% RSLogix 500 project P2a_DIGITAL FILLING STATION STEP METHOD.RSS, saved by version 8.30.00.16 %
PROJECT "PROJECT2"    % processor: Bul.1763 MicroLogix 1100 Series B %

PROGRAM FILES
  LAD 2 "MAIN"  4 rungs
  LAD 3 "IO"  8 rungs  % IO %
  LAD 4 "STEPS"  5 rungs
  LAD 5 "CTRL"  4 rungs

DATA FILES
  O0 OUTPUT  4 elements
  I1 INPUT  6 elements
  S2 STATUS  66 elements
  B3 BINARY  1 elements
  T4 TIMER  1 elements
  C5 COUNTER  1 elements
  R6 CONTROL  1 elements
  N7 INTEGER  1 elements
  F8 FLOAT  1 elements

LADDER 2 "MAIN"
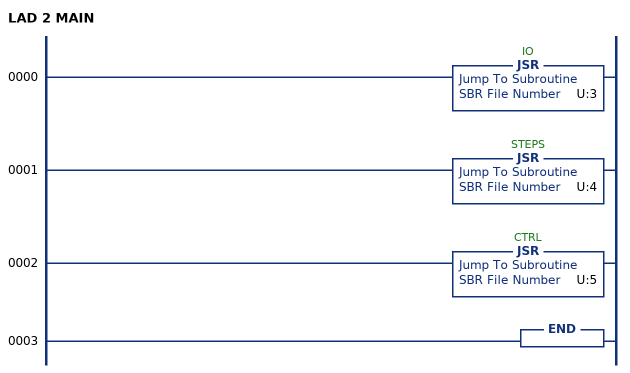
% Rung: 0 %
SOR JSR U:3 EOR
%   U:3  "IO" %
% Rung: 1 %
SOR JSR U:4 EOR
%   U:4  "STEPS" %
% Rung: 2 %
SOR JSR U:5 EOR
%   U:5  "CTRL" %
% Rung: 3 %
SOR END EOR

LADDER 3 "IO"    % IO %
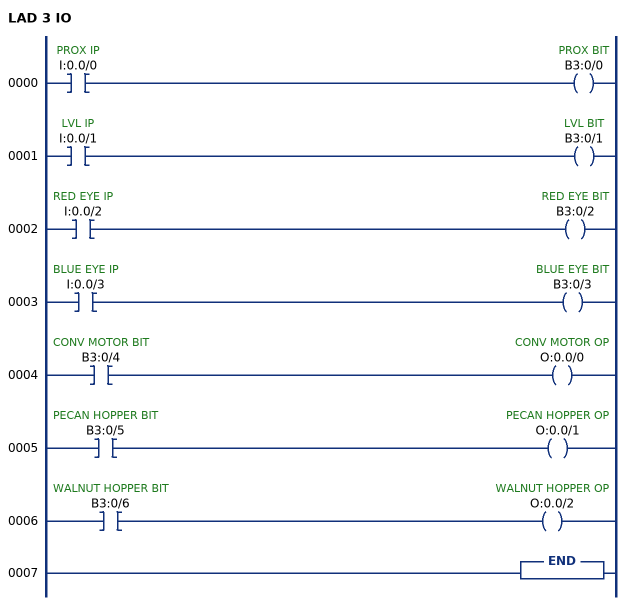
% Rung: 0 %
SOR XIC I:0.0/0 OTE B3:0/0 EOR
%   I:0.0/0  "PROX IP" %
%   B3:0/0  "PROX BIT" %
% Rung: 1 %
SOR XIC I:0.0/1 OTE B3:0/1 EOR
%   I:0.0/1  "LVL IP" %
%   B3:0/1  "LVL BIT" %
% Rung: 2 %
SOR XIC I:0.0/2 OTE B3:0/2 EOR
%   I:0.0/2  "RED EYE IP" %
%   B3:0/2  "RED EYE BIT" %
% Rung: 3 %
SOR XIC I:0.0/3 OTE B3:0/3 EOR
%   I:0.0/3  "BLUE EYE IP" %
%   B3:0/3  "BLUE EYE BIT" %
% Rung: 4 %
SOR XIC B3:0/4 OTE O:0.0/0 EOR
%   B3:0/4  "CONV MOTOR BIT" %
%   O:0.0/0  "CONV MOTOR OP" %
% Rung: 5 %
SOR XIC B3:0/5 OTE O:0.0/1 EOR
%   B3:0/5  "PECAN HOPPER BIT" %
%   O:0.0/1  "PECAN HOPPER OP" %
% Rung: 6 %
SOR XIC B3:0/6 OTE O:0.0/2 EOR
%   B3:0/6  "WALNUT HOPPER BIT" %
%   O:0.0/2  "WALNUT HOPPER OP" %
% Rung: 7 %
SOR END EOR

LADDER 4 "STEPS"
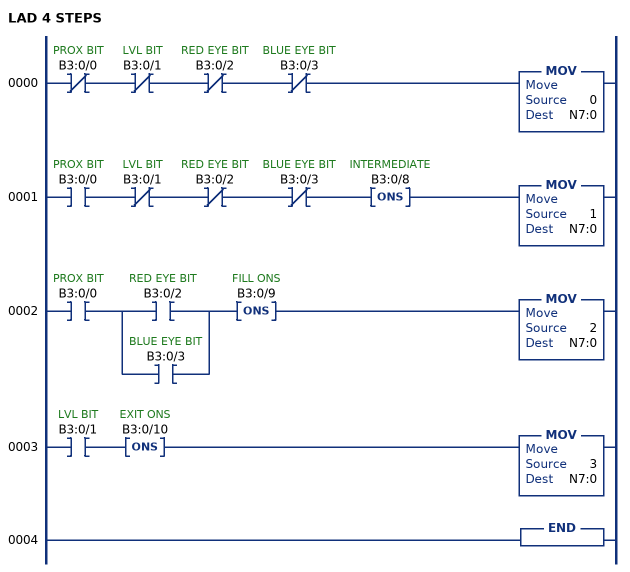
% Rung: 0 %
SOR XIO B3:0/0 XIO B3:0/1 XIO B3:0/2 XIO B3:0/3 MOV 0 N7:0 EOR
%   B3:0/0  "PROX BIT" %
%   B3:0/1  "LVL BIT" %
%   B3:0/2  "RED EYE BIT" %
%   B3:0/3  "BLUE EYE BIT" %
% Rung: 1 %
SOR XIC B3:0/0 XIO B3:0/1 XIO B3:0/2 XIO B3:0/3 ONS B3:0/8 MOV 1 N7:0 EOR
%   B3:0/0  "PROX BIT" %
%   B3:0/1  "LVL BIT" %
%   B3:0/2  "RED EYE BIT" %
%   B3:0/3  "BLUE EYE BIT" %
%   B3:0/8  "INTERMEDIATE" %
% Rung: 2 %
SOR XIC B3:0/0 BST XIC B3:0/2 NXB XIC B3:0/3 BND ONS B3:0/9 MOV 2 N7:0 EOR
%   B3:0/0  "PROX BIT" %
%   B3:0/2  "RED EYE BIT" %
%   B3:0/3  "BLUE EYE BIT" %
%   B3:0/9  "FILL ONS" %
% Rung: 3 %
SOR XIC B3:0/1 ONS B3:0/10 MOV 3 N7:0 EOR
%   B3:0/1  "LVL BIT" %
%   B3:0/10  "EXIT ONS" %
% Rung: 4 %
SOR END EOR

LADDER 5 "CTRL"
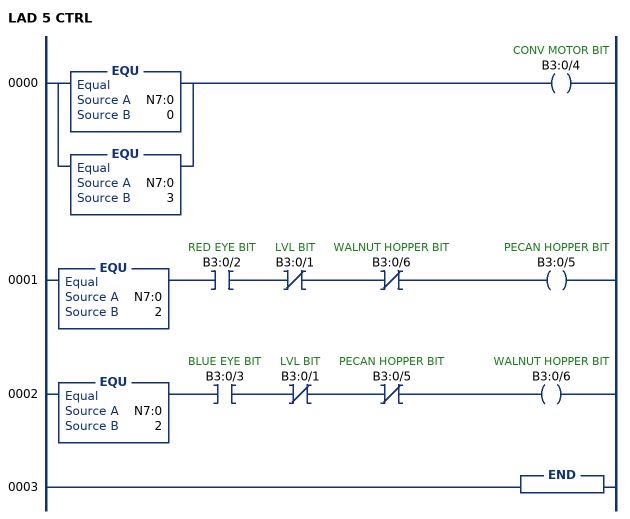
% Rung: 0 %
SOR BST EQU N7:0 0 NXB EQU N7:0 3 BND OTE B3:0/4 EOR
%   B3:0/4  "CONV MOTOR BIT" %
% Rung: 1 %
SOR EQU N7:0 2 XIC B3:0/2 XIO B3:0/1 XIO B3:0/6 OTE B3:0/5 EOR
%   B3:0/2  "RED EYE BIT" %
%   B3:0/1  "LVL BIT" %
%   B3:0/6  "WALNUT HOPPER BIT" %
%   B3:0/5  "PECAN HOPPER BIT" %
% Rung: 2 %
SOR EQU N7:0 2 XIC B3:0/3 XIO B3:0/1 XIO B3:0/5 OTE B3:0/6 EOR
%   B3:0/3  "BLUE EYE BIT" %
%   B3:0/1  "LVL BIT" %
%   B3:0/5  "PECAN HOPPER BIT" %
%   B3:0/6  "WALNUT HOPPER BIT" %
% Rung: 3 %
SOR END EOR

DATA TABLE (non-zero values as saved)
DATA B3
% B3:0 % 0X0010
